{attribute 'qualified_only'}
{attribute 'strict'}
TYPE E_ACTUATOR_RPC_ERROR :
(
	OK						:= 0,
	NOT_OP					:= -1,			
	NOT_NOTOP_READY			:= -2,			
	NOT_NOTOP				:= -3,			
	SWITCHING_ON			:= -4,			
	SWITCHING_OFF			:= -5,			
	LOCAL					:= -7			
);
END_TYPE

(* stored: Version 1.1.0.1, ProductVersion 3.1.4024.3
   DUT E_ACTUATOR_RPC_ERROR: Id {ae0abd72-7773-43bc-83e5-11d973ea74e5} *)
